{attribute 'linkalways'} 
{attribute 'no_explicit_call' := 'This FB is a CLASS and must be accessed using methods or properties'}
{attribute 'enable_dynamic_creation'}
FUNCTION_BLOCK _ETcVnSolvePnPMethod EXTENDS EnumDatatypeBase
VAR
	localData : ETcVnSolvePnPMethod;
	activeData : REFERENCE TO ETcVnSolvePnPMethod;
	enumBaseDatatype : _DINT(localData);
END_VAR

METHOD PRIVATE AddLocalEnumeration
VAR_INPUT
	Enumeration : T_MAXSTRING;
	Value : ETcVnSolvePnPMethod;
END_VAR
AddEnumeration(Enumeration, Value);
END_METHOD

PROPERTY PUBLIC Address : PVOID
GET
Address := ADR(activeData);
END_GET
END_PROPERTY

METHOD PUBLIC ClearReference
VAR_INPUT
END_VAR
activeData REF= localData;
SetBaseDatatypeReference();
END_METHOD

METHOD PUBLIC Clone : I_Datatype
VAR
    pClone : POINTER TO _ETcVnSolvePnPMethod;
END_VAR
pClone := __NEW(_ETcVnSolvePnPMethod(InitialValue := Value));
Clone := pClone^;
END_METHOD

METHOD FB_init : BOOL
VAR_INPUT
	bInitRetains : BOOL; // if TRUE, the retain variables are initialized (warm start / cold start)
	bInCopyCode : BOOL;  // if TRUE, the instance afterwards gets moved into the copy code (online change)
	InitialValue : ETcVnSolvePnPMethod;
END_VAR
localData := InitialValue;
AddBaseDatatype(enumBaseDatatype);
ClearReference();

AddLocalEnumeration('TCVN_SPM_ITERATIVE', ETcVnSolvePnPMethod.TCVN_SPM_ITERATIVE);
AddLocalEnumeration('TCVN_SPM_EPNP', ETcVnSolvePnPMethod.TCVN_SPM_EPNP);
AddLocalEnumeration('TCVN_SPM_P3P', ETcVnSolvePnPMethod.TCVN_SPM_P3P);
AddLocalEnumeration('TCVN_SPM_AP3P', ETcVnSolvePnPMethod.TCVN_SPM_AP3P);
AddLocalEnumeration('TCVN_SPM_IPPE', ETcVnSolvePnPMethod.TCVN_SPM_IPPE);
AddLocalEnumeration('TCVN_SPM_IPPE_SQUARE', ETcVnSolvePnPMethod.TCVN_SPM_IPPE_SQUARE);
AddLocalEnumeration('TCVN_SPM_SQPNP', ETcVnSolvePnPMethod.TCVN_SPM_SQPNP);
END_METHOD

PROPERTY PUBLIC Identifier : T_MAXSTRING
GET
Identifier := 'ETcVnSolvePnPMethod';
END_GET
END_PROPERTY

METHOD IsEnumeratorValueEqual : BOOL
VAR_INPUT
	Enumerator : I_KeyValueForwardEnumerator;
END_VAR
VAR
	storedValue : ETcVnSolvePnPMethod;
END_VAR
IF NOT Enumerator.TryGet(storedValue) THEN
	RETURN;
END_IF

IsEnumeratorValueEqual := storedValue = activeData;
END_METHOD

METHOD PUBLIC MakeReferenceTo
VAR_INPUT
	ReferenceTarget : REFERENCE TO ETcVnSolvePnPMethod;
END_VAR
activeData REF= ReferenceTarget;
SetBaseDatatypeReference();
END_METHOD

METHOD PROTECTED SetBaseDatatypeReference
VAR_INPUT
END_VAR
enumBaseDatatype.MakeReferenceTo(activeData);
END_METHOD

PROPERTY PUBLIC Size : UDINT
GET
Size := SIZEOF(activeData);
END_GET
END_PROPERTY

METHOD TryMakeReferenceTo : BOOL
VAR_INPUT
	Target : I_Datatype;
END_VAR
VAR
	targetAsEnum : I_EnumDatatype;
	pTargetData : POINTER TO ETcVnSolvePnPMethod;
END_VAR
IF NOT Target.TryResolveAsEnumDatatype(targetAsEnum) THEN
	RETURN;
END_IF

IF targetAsEnum.Identifier <> Identifier THEN
	RETURN;
END_IF

pTargetData := Target.Address;
activeData REF= pTargetData^;
SetBaseDatatypeReference();
TryMakeReferenceTo := TRUE;
END_METHOD

PROPERTY PUBLIC Value : ETcVnSolvePnPMethod
GET
Value := activeData;
END_GET
SET
activeData := Value;
END_SET
END_PROPERTY

END_FUNCTION_BLOCK

(* stored: Version 1.1.0.1, ProductVersion 3.1.4024.12
   POU _ETcVnSolvePnPMethod: Id {09e33712-f1dc-418b-abd6-9d0c12aa2cd0}, SpecialFunc None
   Folder Constructor: Id {7bec12f8-202e-482b-8dc0-4feaa1a5bd2d}
   Folder Private: Id {977b3a90-7035-4a04-a53b-01f1afb13a4b}
   Folder Protected: Id {33b9dbd5-7e99-4f8d-9cbc-290e5fc93424}
   Method AddLocalEnumeration: Id {eb82f0cf-ce83-4373-a05a-4620c427be11}
   Property Address: Id {06495e49-a60e-4170-b7d4-865bc579494a}
   Get Get: Id {2f630b28-0a65-4c82-a505-44dafbad7d44}
   Method ClearReference: Id {e2875eca-ebe8-4b10-8673-4e4fab37e8f2}
   Method Clone: Id {a8101c9c-fc8d-44cd-9902-d09d1121103f}
   Method FB_init: Id {81b0bb1d-c098-4663-bca1-bf81ace61f67}
   Property Identifier: Id {d03fd843-69e3-4f2a-8669-74361265bccb}
   Get Get: Id {ee048062-3c48-4720-b468-944d8ec2f344}
   Method IsEnumeratorValueEqual: Id {79ef74b0-0ae3-42df-96f9-0e64625d4fb4}
   Method MakeReferenceTo: Id {d8580204-88a6-42a4-bf77-4c51492e86dc}
   Method SetBaseDatatypeReference: Id {642bb32b-a93d-4248-95e5-d2962bf15955}
   Property Size: Id {a15e31c3-c2cd-4865-8b5d-b301c7f42453}
   Get Get: Id {73ce94f4-9069-4b74-a9d1-da86d0dee865}
   Method TryMakeReferenceTo: Id {d0ca4815-38c1-4c4c-912e-56c291f76f27}
   Property Value: Id {bf8b7a9c-c335-4e63-915a-7bd149c880a7}
   Get Get: Id {b8955399-a94f-4ffa-ae17-34e2cfa9e7e5}
   Set Set: Id {6d4f359a-bfc6-4008-87d0-3f4714009446} *)
